// TIA Portal V20 export
ORGANIZATION_BLOCK "CyclicInterrupt"   // OB33, LAD, CyclicInterrupt
// stored: Namespace Unit1.Em3, SetENOAutomatically false
   VAR_INPUT
      Initial_Call : Bool;   // Initial call of this OB
      Event_Count : Int;   // Events discarded
   END_VAR
BEGIN
END_ORGANIZATION_BLOCK
